(* IEC 61131-3 sources: plc_on_fpga_riscv_hybrid/RV_FPGA_PLC_IDE_Projects/PWM_Test, 1 file *)

(* ---- PWM_Test.il ---- *)
VAR
    PWM_1   : PWM
END_VAR

PROGRAM PWM_Test
    R1 :
        CAL PWM_1(
            F  := 2,
            DC := 80,
            Q  => %LEDG.0)
END_PROGRAM
